{attribute 'GeneratedUsingTerminal: KL6401-0002'}
{attribute addProperty BoxType "KL6401-0002"}
{attribute addProperty Id "Parameter_StatusAT %I*UINT0Parameter_Input_Data_1AT %I*UDINT0Parameter_Input_Data_2AT %I*UDINT0Parameter_Input_Data_3AT %I*UDINT0Parameter_Input_Data_4AT %I*UDINT0Parameter_Input_Data_5AT %I*UDINT0Parameter_Input_Data_6AT %I*UDINT0Parameter_Input_Data_7AT %I*UDINT0Parameter_Input_Data_8AT %I*UDINT0Parameter_TypeAT %I*USINT0LON_StatusAT %I*USINT0Parameter_ControlAT %Q*UINT0Parameter_Output_Data_1AT %Q*UDINT0Parameter_Output_Data_2AT %Q*UDINT0Parameter_Output_Data_3AT %Q*UDINT0Parameter_Output_Data_4AT %Q*UDINT0Parameter_Output_Data_5AT %Q*UDINT0Parameter_Output_Data_6AT %Q*UDINT0Parameter_Output_Data_7AT %Q*UDINT0Parameter_Output_Data_8AT %Q*UDINT0CMDAT %Q*USINT0IdxAT %Q*USINT0"}
{attribute addProperty CRC "1980160393"}
{attribute addProperty Size "0"}
TYPE Channel_7606D989 :
STRUCT
	{attribute addProperty Name "Parameter_Status"}
	Parameter_Status AT %I* : UINT;
	{attribute addProperty Name "Parameter_Input_Data_1"}
	Parameter_Input_Data_1 AT %I* : UDINT;
	{attribute addProperty Name "Parameter_Input_Data_2"}
	Parameter_Input_Data_2 AT %I* : UDINT;
	{attribute addProperty Name "Parameter_Input_Data_3"}
	Parameter_Input_Data_3 AT %I* : UDINT;
	{attribute addProperty Name "Parameter_Input_Data_4"}
	Parameter_Input_Data_4 AT %I* : UDINT;
	{attribute addProperty Name "Parameter_Input_Data_5"}
	Parameter_Input_Data_5 AT %I* : UDINT;
	{attribute addProperty Name "Parameter_Input_Data_6"}
	Parameter_Input_Data_6 AT %I* : UDINT;
	{attribute addProperty Name "Parameter_Input_Data_7"}
	Parameter_Input_Data_7 AT %I* : UDINT;
	{attribute addProperty Name "Parameter_Input_Data_8"}
	Parameter_Input_Data_8 AT %I* : UDINT;
	{attribute addProperty Name "Parameter_Type"}
	Parameter_Type AT %I* : USINT;
	{attribute addProperty Name "LON_Status"}
	LON_Status AT %I* : USINT;
	{attribute addProperty Name "Parameter_Control"}
	Parameter_Control AT %Q* : UINT;
	{attribute addProperty Name "Parameter_Output_Data_1"}
	Parameter_Output_Data_1 AT %Q* : UDINT;
	{attribute addProperty Name "Parameter_Output_Data_2"}
	Parameter_Output_Data_2 AT %Q* : UDINT;
	{attribute addProperty Name "Parameter_Output_Data_3"}
	Parameter_Output_Data_3 AT %Q* : UDINT;
	{attribute addProperty Name "Parameter_Output_Data_4"}
	Parameter_Output_Data_4 AT %Q* : UDINT;
	{attribute addProperty Name "Parameter_Output_Data_5"}
	Parameter_Output_Data_5 AT %Q* : UDINT;
	{attribute addProperty Name "Parameter_Output_Data_6"}
	Parameter_Output_Data_6 AT %Q* : UDINT;
	{attribute addProperty Name "Parameter_Output_Data_7"}
	Parameter_Output_Data_7 AT %Q* : UDINT;
	{attribute addProperty Name "Parameter_Output_Data_8"}
	Parameter_Output_Data_8 AT %Q* : UDINT;
	{attribute addProperty Name "CMD"}
	CMD AT %Q* : USINT;
	{attribute addProperty Name "Idx"}
	Idx AT %Q* : USINT;
END_STRUCT
END_TYPE

(* stored: Version 1.2.0.0, ProductVersion 3.1.4024.9
   DUT Channel_7606D989: Id {b43eb2af-d7db-4885-ab35-05c5a43e712b} *)
